% RSLogix 500 project NEGABS.RSS, saved by version 9.00.00.04 %
PROJECT "UNTITLED"    % processor: Bul.1763 MicroLogix 1100 Series B %

PROGRAM FILES
  LAD 2   3 rungs

DATA FILES
  O0 OUTPUT  4 elements
  I1 INPUT  6 elements
  S2 STATUS  66 elements
  B3 BINARY  1 elements
  T4 TIMER  1 elements
  C5 COUNTER  1 elements
  R6 CONTROL  1 elements
  N7 INTEGER  3 elements
  F8 FLOAT  1 elements
  ST9 STRINGS  4 elements

LADDER 2
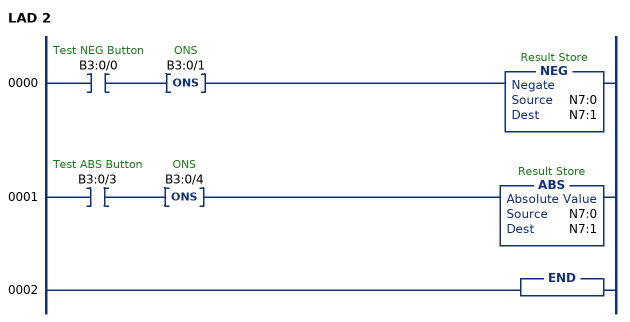
% Rung: 0 %
SOR XIC B3:0/0 ONS B3:0/1 NEG N7:0 N7:1 EOR
%   B3:0/0  "Test NEG Button" %
%   B3:0/1  "ONS" %
%   N7:0  "0 = FALSE 1 = TRUE" %
%   N7:1  "Result Store" %
% Rung: 1 %
SOR XIC B3:0/3 ONS B3:0/4 ABS N7:0 N7:1 EOR
%   B3:0/3  "Test ABS Button" %
%   B3:0/4  "ONS" %
%   N7:0  "0 = FALSE 1 = TRUE" %
%   N7:1  "Result Store" %
% Rung: 2 %
SOR END EOR

OTHER DOCUMENTED ADDRESSES
  B3:0/2  "Test ACN Trigger Bit"
  B3:0/5  "Test ASR Trigger Bit"
  ST9:0  "Partial String 1"
  ST9:1  "Partial String 2"
  ST9:2  "Concatenated String"
  ST9:3  "Test Value"

DATA TABLE (non-zero values as saved)
DATA ST9
% ST9:0 % "TEST"
% ST9:1 % "STRING"
% ST9:2 % "SOMETHING"
% ST9:3 % "TESTSTRING"
